FUNCTION_BLOCK EV_StopperArm (* Typed view of StopperArm's state channel (inputs and holder) *)
  (* Standard: 61499-2 *)
  (* Version 0.1, 2026-09-28, Project contributors, AAU Smart Production Lab *)
  PACKAGE stoppering;
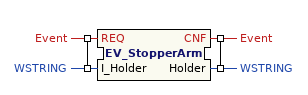
  EVENT_INPUT
    REQ WITH I_Holder;
  END_EVENT
  EVENT_OUTPUT
    CNF WITH Holder;
  END_EVENT
  VAR_INPUT
    I_Holder : WSTRING;
  END_VAR
  VAR_OUTPUT
    Holder : WSTRING;
  END_VAR
  EC_STATES
    REQ : REQ -> CNF;
  END_STATES
  ALGORITHM REQ IN ST:
Holder := I_Holder;
  END_ALGORITHM
END_FUNCTION_BLOCK
